(*======================================================================================================================================*)
(*RS485_COM_PRG: Beispielhaftes Programm zum Steuern von HAus-Bus.de Komponenten über RS485 mit TwinCAT
					Achtung dieser POU muss als 1ms Task Aufgerufen werden um Ordnungsgemäß zu laufen *)
(*
Date          	| Version    	| created under        	| Author          	| Remark *)
(*====================================================================================================================================================*)
(*15/05/2025   	| 1.00      		| TC3		  		| N.Kersting       | first release *)
(*====================================================================================================================================================*)

PROGRAM RS485_COM_PRG
VAR  
     i,h,j						:INT;
	
	fbRS485Startup				:fb_RS485Startup;		(* Startup Parametrierung der Klemme/ RS485 Bus *)
	fbRS485SendCmdFiFo			:fb_RS485FiFoMaster;	(* Sende und Empfangs FiFo für RS485 *)
	fbLineControl 				:SerialLineControl;		(* Hält die Serielle Kommunikation Aufrecht *)
	
	fComBufferReset				:ClearComBuffer;		(* Löschen des SPS Internen Bufferinhalts *)
	
	rxBuffer 					:ComBuffer;				(* COM Buffer Empfangen *)
    txBuffer 					:ComBuffer;				(* COM Buffer Senden *)
	
	
END_VAR

(* IDs Setzen *)
ac00_HausBusIdRS485COM();
(* RS485 Klemmen Config *)
ac01_StartupRS485COM();

ACTION ac00_HausBusIdRS485COM:
(* Initialisierung der Gerätenamen *)
(* Achtung nur Beispiele *)
stHBDeviceIdent[1].sName	:=			'Wohnzimmer';
stHBDeviceIdent[1].diID	:=				5256;
stHBDeviceIdent[1].sPingIdent :=		'TMP.1.gSTATUS';

stHBDeviceIdent[2].sName	:=			'Test1';
stHBDeviceIdent[2].diID	:=				5269;
stHBDeviceIdent[2].sPingIdent :=		'TMP.1.gSTATUS';

stHBDeviceIdent[3].sName	:=			'Test2';
stHBDeviceIdent[3].diID	:=				1234;
stHBDeviceIdent[3].sPingIdent :=		'TMP.1.gSTATUS';

stHBDeviceIdent[4].sName	:=			'Test3';
stHBDeviceIdent[4].diID	:=				3333;
stHBDeviceIdent[4].sPingIdent :=		'TMP.1.gSTATUS';

stHBDeviceIdent[5].sName	:=			'Test4';
stHBDeviceIdent[5].diID	:=				4444;
stHBDeviceIdent[5].sPingIdent :=		'TMP.1.gSTATUS';

stHBDeviceIdent[6].sName	:=			'';
stHBDeviceIdent[6].diID	:=				0;
stHBDeviceIdent[6].sPingIdent :=		'TMP.1.gSTATUS';

stHBDeviceIdent[7].sName	:=			'';
stHBDeviceIdent[7].diID	:=				0;
stHBDeviceIdent[7].sPingIdent :=		'TMP.1.gSTATUS';

stHBDeviceIdent[8].sName	:=			'';
stHBDeviceIdent[8].diID	:=				0;
stHBDeviceIdent[8].sPingIdent :=		'TMP.1.gSTATUS';

stHBDeviceIdent[9].sName	:=			'';
stHBDeviceIdent[9].diID	:=				0;
stHBDeviceIdent[9].sPingIdent :=		'TMP.1.gSTATUS';

stHBDeviceIdent[10].sName	:=			'';
stHBDeviceIdent[10].diID	:=			0;
stHBDeviceIdent[10].sPingIdent :=		'TMP.1.gSTATUS';

stHBDeviceIdent[11].sName	:=			'Jalousie 1';
stHBDeviceIdent[11].diID	:=			5614;
stHBDeviceIdent[11].sPingIdent :=		'OUT.210.gSTATUS';

stHBDeviceIdent[12].sName	:=			'';
stHBDeviceIdent[12].diID	:=			0;
stHBDeviceIdent[12].sPingIdent :=		'OUT.210.gSTATUS';

stHBDeviceIdent[13].sName	:=			'CYD Test';
stHBDeviceIdent[13].diID	:=			5999;
stHBDeviceIdent[13].sPingIdent :=		'OUT.210.gSTATUS';
END_ACTION

ACTION ac01_StartupRS485COM:

(* Klemmen Startup, inkl Klemmenkonfiguration usw. *)
fbRS485Startup(
	I_bExecute:= 		TRUE, 
	I_bBusOK:= 			uiEtherCATStateBK1120_RS485COM = 8
						AND uiKBusStateBK1120_RS485COM = 0, 
	I_tStartupVerz:= 	T#5S, 
	IQ_InData:= 		KL6041In, 
	IQ_OutData:= 		KL6041Out, 
	Q_sState=> , 
	Q_bStartupDone=> , 
	Q_bError=> );

(* Aktivierung der Linecontrole erst wenn Startup erfolgt *)	
IF fbRS485Startup.Q_bStartupDone
THEN
	fbLineControl(
		Mode := 		ComSerialLineMode_t.SERIALLINEMODE_KL6_22B_STANDARD,
		pComIn := 		ADR(KL6041In),
		pComOut := 		ADR(KL6041Out),
		SizeComIn := 	UINT_TO_INT(SIZEOF(KL6041In)),
		RxBuffer := 	rxBuffer,
		TxBuffer := 	txBuffer );
				
	(* Relais *)
	ac10_HausBusRelaisRS485COM();
	(* Taster *)
	ac10_HausBusTasterRS485COM();
	(* CYD *)
	ac10_HausBusCYDRS485COM();
	
	
	(* Senden FiFo *)			
	fbRS485SendCmdFiFo(
		I_sSendCmdFiFo:= 		GVL_RS485FiFoSend.sSendFiFo, 
		I_stDeviceIdent :=		stHBDeviceIdent,
		I_bAutoPing:= 			bUseFiFoPing, 
		I_tAutoPingTime:= 		cPingSendTimeFiFo,		 
		I_bManuellMode:= 		, 
		I_sSendCmdManuell:= 	, 
		I_bSendManuell:= 		, 
		I_bExecute:= 			TRUE, 
		I_bBusBelastungstest:= 	, 
		I_bReset:= 				, 
		I_sStartZeichen:= 		, 
		I_sEndZeichen:= 		, 
		I_pTxBuffer:= 			ADR(txBuffer), 
		I_pRxBuffer:= 			ADR(rxBuffer), 
		Q_sReceiveString=> , 
		Q_lrBusAuslastung=> , 
		Q_bBusy=> , 
		Q_bDone=> , 
		Q_bError=> , 
		Q_sState=> , 
		Q_stStates=> );
		
ELSE
	(* Com Buffer zum Resetten *)
	fComBufferReset(Buffer:= rxBuffer);
	fComBufferReset(Buffer:= txBuffer);
END_IF
END_ACTION

ACTION ac10_HausBusCYDRS485COM:
(* Bustaster Aufrufe *)
FOR j := cMaxBusRelais+cMaxBusTaster+2 TO cMaxBusRelais+cMaxBusTaster+cMaxCYD+1 BY 1 DO
		
	fbCYDHB6F[j].I_stInput.sName :=	stHBDeviceIdent[j].sName;
	fbCYDHB6F[j].I_stInput.diID	:=	stHBDeviceIdent[j].diID;
	
	IF GVL_ServiceVisu.bCYDServiceAktiv[j]
	THEN
		fbCYDHB6F[j].I_stInput.iLED := GVL_ServiceVisu.stCYDService[j].iLED;
		fbCYDHB6F[j].I_stInput.iLEDBg := GVL_ServiceVisu.stCYDService[j].iLEDBg;
		fbCYDHB6F[j].I_stInput.iLEDExt := GVL_ServiceVisu.stCYDService[j].iLEDExt;
		fbCYDHB6F[j].I_stInput.bReset := GVL_ServiceVisu.stCYDService[j].bReset;
		fbCYDHB6F[j].I_stInput.bServiceMode := GVL_ServiceVisu.stCYDService[j].bServiceMode;
		fbCYDHB6F[j].I_stInput.bService := GVL_ServiceVisu.stCYDService[j].bService;
		fbCYDHB6F[j].I_stInput.bWifi := GVL_ServiceVisu.stCYDService[j].bWifi;
		fbCYDHB6F[j].I_stInput.bWebServer := GVL_ServiceVisu.stCYDService[j].bWebServer;
		
	END_IF
	
	stCYDService[j].sName :=	fbCYDHB6F[j].I_stInput.sName;
	stCYDService[j].diID :=		fbCYDHB6F[j].I_stInput.diID;
	
	fbCYDHB6F[j].I_stInput.bExecute := TRUE;
	fbCYDHB6F[j](
		I_FifoID :=			j,
		I_bPingStart:= 		TRUE , 	(* Taster Verzögert Pingen, damit weniger Busauslastung entsteht *)
		I_StringReceived:=	fbRS485SendCmdFiFo.Q_sReceiveString);
		
	(* Sendebefehle an FiFo Übergeben *)
	GVL_RS485FiFoSend.sSendFiFo[j] :=	fbCYDHB6F[j].Q_sFiFoSend;
END_FOR
END_ACTION

ACTION ac10_HausBusRelaisRS485COM:
(* BusRelais Aufrufe *)
FOR h := cMaxBusTaster +1 TO cMaxBusRelais+cMaxBusTaster+1 BY 1 DO (*cMaxBusTaster+1..cMaxBusRelais+cMaxBusTaster+1*)
		
	fbRelaisHB16F[h].I_stInput.sName :=	stHBDeviceIdent[h].sName;
	fbRelaisHB16F[h].I_stInput.diID	:=	stHBDeviceIdent[h].diID;
	
	IF GVL_ServiceVisu.bRelaisServiceAktiv[h]
	THEN
		fbRelaisHB16F[h].I_stInput.bOut := stRelaisService[h].bOut;
		fbRelaisHB16F[h].I_stInput.bReset := stRelaisService[h].bReset;
	END_IF
	
	stRelaisService[h].sName :=	fbRelaisHB16F[h].I_stInput.sName;
	stRelaisService[h].diID :=	fbRelaisHB16F[h].I_stInput.diID;
	
	fbRelaisHB16F[h].I_stInput.bExecute := TRUE;
	fbRelaisHB16F[h](
		I_FifoID :=			h,
		I_bPingStart:= 		TRUE,	(* Direkt Starten *)
		I_StringReceived:=	fbRS485SendCmdFiFo.Q_sReceiveString);
		
	(* Sendebefehle an FiFo Übergeben *)
	GVL_RS485FiFoSend.sSendFiFo[h] :=	fbRelaisHB16F[h].Q_sFiFoSend;	
END_FOR
END_ACTION

ACTION ac10_HausBusTasterRS485COM:
(* Bustaster Aufrufe *)
FOR i := 1 TO cMaxBusTaster BY 1 DO
			
	fbTasterHB6F[i].I_stInput.sName :=	stHBDeviceIdent[i].sName;
	fbTasterHB6F[i].I_stInput.diID	:=	stHBDeviceIdent[i].diID;
	
	IF GVL_ServiceVisu.bTasterServiceAktiv[i]
	THEN
		fbTasterHB6F[i].I_stInput.iLED := GVL_ServiceVisu.stTasterService[i].iLED;
		fbTasterHB6F[i].I_stInput.iLEDBg := GVL_ServiceVisu.stTasterService[i].iLEDBg;
		fbTasterHB6F[i].I_stInput.iLEDExt := GVL_ServiceVisu.stTasterService[i].iLEDExt;
		fbTasterHB6F[i].I_stInput.bReset := GVL_ServiceVisu.stTasterService[i].bReset;
	END_IF
	
	stTasterService[i].sName :=	fbTasterHB6F[i].I_stInput.sName;
	stTasterService[i].diID :=	fbTasterHB6F[i].I_stInput.diID;
	
	fbTasterHB6F[i].I_stInput.bExecute := TRUE;
	fbTasterHB6F[i](
		I_FifoID :=			i,
		I_bPingStart:= 		TRUE , 	(* Taster Verzögert Pingen, damit weniger Busauslastung entsteht *)
		I_StringReceived:=	fbRS485SendCmdFiFo.Q_sReceiveString);
		
	(* Sendebefehle an FiFo Übergeben *)
	GVL_RS485FiFoSend.sSendFiFo[i] :=	fbTasterHB6F[i].Q_sFiFoSend;
END_FOR
END_ACTION

END_PROGRAM

(* stored: Version 1.1.0.1, ProductVersion 3.1.4024.12
   POU RS485_COM_PRG: Id {6dd6665a-a6d4-412f-b9c4-7cb94f6da62e}, SpecialFunc None
   Folder Aufrufe: Id {6e56fed8-3c26-47a0-8e19-67d3f91b47b1}
   Action ac00_HausBusIdRS485COM: Id {5732253f-e0f1-4a17-91db-75baa6756837}
   Action ac01_StartupRS485COM: Id {354e2a31-8e9f-4c62-8bef-dabbbf0da490}
   Action ac10_HausBusCYDRS485COM: Id {1feac4c3-8270-47f7-bbe2-dba512bcd624}
   Action ac10_HausBusRelaisRS485COM: Id {c08d890d-e2db-478d-a692-045466c2ee35}
   Action ac10_HausBusTasterRS485COM: Id {f4fb0d91-a1c4-466e-8327-78f0013f7848} *)
